function_block FB_Syntax_Pragmas
VAR  
    nValue : int;  
end_var

{region 'Init'}  
nValue := 1;
{endregion}  


{formatting.disable}
nValue := 99;
{formatting.enable}

END_FUNCTION_BLOCK

(* stored: Version 1.1.0.1, ProductVersion 3.1.4024.16
   POU FB_Syntax_Pragmas: Id {fa333a5b-3b1c-45b4-adaa-60a93a52ba05}, SpecialFunc None *)
